FUNCTION_BLOCK F_AnzeigeSollpositionsFehler 
VAR_INPUT
	enable : BOOL;
	errNo : WORD;
	idOffset : WORD; 
END_VAR
VAR_OUTPUT
	errID : WORD;
END_VAR
VAR
	//wait : TON;
END_VAR

errID := idOffset;
IF enable THEN
	
	//wait(IN := errNo > 0, PT := T#1S);
	//IF wait.Q THEN
		errID := idOffset + errNo;
	//END_IF

END_IF

END_FUNCTION_BLOCK

(* stored: Version 1.1.0.1, ProductVersion 3.1.4024.3
   POU F_AnzeigeSollpositionsFehler: Id {21cf8165-5988-47a9-814a-3a4fb28a144a}, SpecialFunc None *)
